Staubli VAL3: page_simulation.pjx

--- page_simulation.pjx ---
Parameters version=s7.5 stackSize=5000 millimeterUnit=true
Program file=CycleRefresh.pgx
Program file=goTo.pgx
Program file=isAtPoint.pgx
Program file=loadEditTraj.pgx
Program file=loadPage.pgx
Program file=loadType.pgx
Program file=main.pgx
Program file=onEnterEvent.pgx
Program file=onExit.pgx
Program file=onF1Event.pgx
Program file=onF2Event.pgx
Program file=onF3Event.pgx
Program file=onF4Event.pgx
Program file=onF5Event.pgx
Program file=onF6Event.pgx
Program file=onF7Event.pgx
Program file=onF8Event.pgx
Program file=onStart.pgx
Program file=printToShow.pgx
Program file=refresh.pgx
Program file=refreshDynamic.pgx
Program file=refreshPoints.pgx
Program file=refreshStatic.pgx
Program file=showMessage.pgx
Program file=startCycle.pgx
Program file=stepping.pgx
Program file=stopCycle.pgx
Data file=page_simulation.dtx
Library alias=page path=Disk://kernel/template/page/page.pjx
Library alias=use path=Disk://kernel/userPage/userPage.pjx
Library alias=language path=Disk://kernel/language/language.pjx
Library alias=saveData path=Disk://saveData/saveData.pjx
Library alias=cycleStatus path=Disk://cycleStatus/cycleStatus.pjx
Library alias=trajType path=Disk://../templates/trajectory/trajectory.pjx
Library alias=OnEvent path=Disk://OnEvent/OnEvent.pjx
Type name=TrajectoryItem path=Disk://kernel/template/TrajectoryItem/TrajectoryItem.pjx
Type name=InstrItem path=Disk://kernel/template/InstrItem/InstrItem.pjx

--- isAtPoint.pgx ---
program isAtPoint(num x_nIndex, bool& x_bInside[])
  local point l_pHere
  local tool l_tTool
  local num l_nDistance
  local point l_pPoint[2]
  local num l_nIndexTool
  local TrajectoryItem l_tTrajItem
begin
  // reset the bool
  x_bInside=false
  // get the tcp
  call trajType:getTool(l_nIndexTool)
  call saveData:getTool(l_tTool,l_nIndexTool)
  // get the mdesc
  call trajType:getTrajItem(l_tTrajItem,x_nIndex)
  // get the acutal point
  l_pHere=here(l_tTool,world)
  // look if the robot is inside the blend area
  call trajType:getPoint(l_pPoint,false,x_nIndex)
  // check the radius
  if distance(position(l_pPoint,world),l_pHere.trsf)<=max(l_nDistance,nRoundStepping)
    x_bInside=true
  endIf
end

--- loadEditTraj.pgx ---
program loadEditTraj(string x_sName)
  local num i
begin
  // load the type
  call trajType:load(x_sName,i)
  if i!=0
    popUpMsg("Loading trajectory type "+x_sName+" error CODE "+toString("",i))
    logMsg("INTERFACE:TRAJECTORY LIBLOAD "+x_sName+" result "+toString("",i))
  endIf
end

--- loadPage.pgx ---
program loadPage(string x_sPage, string& x_sItems[])
// load the next page
  local num i
  local string l_sMessage
begin
  // look if the page libload is correct
  i=page:libLoad(x_sPage)
  delay(0)
  if i!=0
    logMsg("[KERNEL] INTERFACE:PAGE LIBLOAD "+x_sPage+" result "+toString("",i))
    call language:message(l_sMessage,-7)
    popUpMsg(l_sMessage+x_sPage+" ; "+toString("",i))
  else
    // copy all the field from x_sItems to the next page
    call use:stringCopy(x_sItems,page:sItems)
    call page:main()
    // to give back
    call use:stringCopy(page:sItems,x_sItems)
    //
    bShowMessage=false
    use:bUseRefresh=true
  endIf
end

--- loadType.pgx ---
program loadType(num& x_nResult[])
  local num i
  local num l_nIndex
  local string l_sPath
begin
  if find(trajType:libPath(),saveData:sTrajTypeUsing)==-1
    // load the traj type
    call saveData:getPathInstr(saveData:sTrajTypeUsing,l_sPath)
    x_nResult=trajType:libLoad(l_sPath)
    delay(0)
    if x_nResult!=0
      popUpMsg("error load traj type on START "+saveData:sTrajTypeUsing+toString("",x_nResult))
    endIf
  endIf
end

--- onEnterEvent.pgx ---
program onEnterEvent()
  local num l_nPoint
  local bool l_bInside
  local bool l_bOk
begin
  //
  // NB sEvent is the selected
  // element in the LIST
  //
  if !cycleStatus:bSimulation
    call use:stringToArray(sTrajName+","+toString("",nPoint),sMessage)
    // reload the traj
    //call loadEditTraj(sTrajName)
    //
    call loadPage("Disk://trajectory/page_editTraj",sMessage)
    // reload the traj
    call loadEditTraj(sTrajName)
    //
    // ELEBORATE THE GIVE BACK
    //
    l_bOk=true
    toNum(sMessage[1],l_nPoint,l_bOk)
    call isAtPoint(l_nPoint,l_bInside)
    if l_bInside
      nPoint=l_nPoint
    endIf
    cls()
    use:bUseRefresh=true
    // reset the show status
    bShowStatus=false
  endIf
end

--- onF1Event.pgx ---
program onF1Event()
  local num l
begin
  // look if the bButton is enable
  if bButton[0]
    //
    // go to previous POINT
    //
    if !cycleStatus:bCycle or !cycleStatus:bSimulation
      call goTo(nPoint-1)
    endIf
  endIf
end

--- onF2Event.pgx ---
program onF2Event()
  local tool l_tTool
  local bool l_bContinue
  local num i
  local num l_nSize
begin
  // look if the bButton is enable
  if bButton[1]
    if cycleStatus:bSimulation
      //
      // ENABLE STEPPING
      //
      call trajType:getSizeItem(false,l_nSize)
      if !bStepping and nPoint<(l_nSize-1) and taskStatus("stepping")==-1 and !isEmpty()
        taskCreate "stepping",20,stepping()
      endIf
    else
      //
      // go to actual POINT
      //
      if !cycleStatus:bCycle or !cycleStatus:bSimulation
        call goTo(nPoint)
      endIf
    endIf
  endIf
end

--- onF5Event.pgx ---
program onF5Event()
begin
  // look if the bButton is enable
  if bButton[4]
    //
    //
  endIf
end

--- onF7Event.pgx ---
program onF7Event()
  local string l_sMessage
  local bool l_bContinue
  local bool l_bYes
  local string l_sItem
  local bool l_bInside
begin
  // look if the bButton is enable
  if bButton[6]
    //
    // STOP /START
    //
    if !cycleStatus:bSimulation and nKey!=255
      if nPoint!=0
        // not for the first point
        call isAtPoint(nPoint,l_bInside)
      else
        l_bInside=true
      endIf
      if l_bInside
        // START
        bStepping=false
        call startCycle(nPoint)
      else
        // not at point
        call language:message(l_sMessage,95)
        call use:timerDialog(l_sMessage+toString("",nPoint+1),2)
      endIf
    elseIf cycleStatus:bSimulation
      // STOP CYCLE
      call stopCycle()
      call use:nullKey(nKey)
    endIf
    //
    //
    use:bUseRefresh=true
    //
  endIf
end

--- onStart.pgx ---
program onStart(num x_nResult)
  local bool l_bOk
  local string l_sButton[2]
  local string l_sMessage
  local string l_sPage
  local string l_sItem
begin
  // clean the movement
  if !isEmpty()
    resetMotion()
  endIf
  nPoint=0
  cls()
  bStepping=false
  // save the traj Name
  sTrajName=sItems
  // INIT the resource
  use:bUseRefresh=true
  // load all
  call loadType(x_nResult)
  //
  // look if the trajType has the stepping enable
  //
  if trajType:bStepping
    call loadEditTraj(sTrajName)
    //
    logMsg("[KERNEL] INTERFACE:PAGE Simulation")
  else
    // only start and return
    call language:message(l_sMessage,214)
    call language:getYesNo(l_sButton)
    // ask the yes_no question
    call use:yes_no(l_sMessage,l_sButton,l_bOk)
    if l_bOk
      cycleStatus:iToSuperV.sType=saveData:sTrajTypeUsing
      cycleStatus:iToSuperV.sData=sTrajName
      cycleStatus:nInterfaceToSV=3
      logMsg("[KERNEL] INTERFACE:Simulation of the item: "+saveData:sTrajTypeUsing+" "+sTrajName)
      wait(cycleStatus:nInterfaceToSV==-1)
      // load the production page
      l_sPage="kernel/page/production"
      l_sItem="simulation"
      call loadPage(l_sPage,l_sItem)
      call use:setView(false)
    endIf
    x_nResult=99
  endIf
  //
end

--- refreshPoints.pgx ---
program refreshPoints(string x_sTrajName)
  local num i
  local num l_nSize
  local string l_sEvent
  local TrajectoryItem l_tTraj
begin
  // load the traj
  call use:listcreate(x_sTrajName)
  //
  call trajType:getSizeItem(false,l_nSize)
  for i=0 to l_nSize-1
    call trajType:getTrajItem(l_tTraj,i)
    l_sEvent=toString("2",i+1)+" "+l_tTraj.comment
    call use:listadd(l_sEvent)
  endFor
  //
end

--- startCycle.pgx ---
program startCycle(num x_nPoint)
  local string l_sMessage
  local bool l_bOk
  local num l_nSize
  local string l_sButton[2]
begin
  // START
  watch(cycleStatus:nInterfaceToSV==-1,5)
  // get the question message
  call language:message(l_sMessage,214)
  call language:getYesNo(l_sButton)
  // ask the yes_no question
  call use:yes_no(l_sMessage,l_sButton,l_bOk)
  if l_bOk
    // reSTART??
    call trajType:getSizeItem(false,l_nSize)
    if nPoint==l_nSize-1
      x_nPoint=nPoint=0
    endIf
    // compose with 2 element
    cycleStatus:iToSuperV.sType=saveData:sTrajTypeUsing
    cycleStatus:iToSuperV.sData=sTrajName+","+toString("",x_nPoint)
    // send the command to the SuperV
    cycleStatus:nInterfaceToSV=3
    logMsg("[KERNEL] INTERFACE:Simulation of the item: "+saveData:sTrajTypeUsing+" "+sTrajName)
    // wait the command has been receive
    watch(cycleStatus:nInterfaceToSV==-1,5)
  endIf
end

--- stepping.pgx ---
program stepping()
  local num l_nId
begin
  //
  // ENABLE STEPPING
  //
  bStepping=true
  call use:clear(0,13)
  call use:typeMenu(7,"STOP")
  // wait the start
  wait((cycleStatus:bSimulation and !isEmpty()) or nKey==255 or nKey==277)
  // look if the key STEP has been pressed
  if nKey!=255 or nKey!=277
    // find one
    if cycleStatus:bSimulation and !isEmpty()
      // go stepping
      call cycleStatus:getLastId(l_nId)
      do
        nKey=getKey()
        delay(0)
        // wait the ID stepping
      until ((getMoveId()>=l_nId-0.015+1) or nKey==255 or nKey==277 or !cycleStatus:bSimulation)
      // stepping is finished
      bStepping=false
      // STOP CYCLE
      if cycleStatus:bSimulation
        call stopCycle()
      endIf
      bShowMessage=false
      //
    endIf
  endIf
end

--- stopCycle.pgx ---
program stopCycle()
begin
  //
  // STOP
  //
  stopMove()
  cycleStatus:bToStop=true
  call use:timerDialog(" STOP CYCLE ",1)
  //
  watch(cycleStatus:bToStop==false,1)
end
